RESOURCE_TYPE top
  (* Standard: 61499-2 *)
  (* Version 0.1, 2017-00-25, hpea485, UOA *)
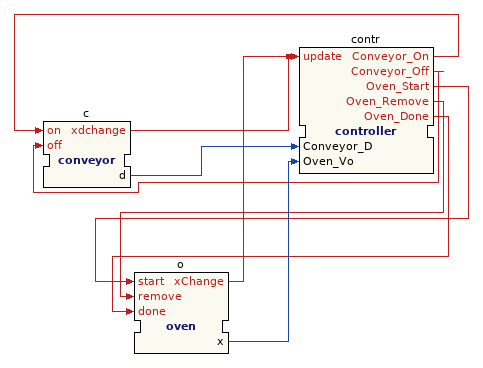
  FBS
    o : oven;
    c : conveyor;
    contr : controller;
  END_FBS
  EVENT_CONNECTIONS
    o.xChange TO contr.update;
    c.xdchange TO contr.update;
    contr.Conveyor_On TO c.on;
    contr.Conveyor_Off TO c.off;
    contr.Oven_Start TO o.start;
    contr.Oven_Remove TO o.remove;
    contr.Oven_Done TO o.done;
  END_CONNECTIONS
  DATA_CONNECTIONS
    o.x TO contr.Oven_Vo;
    c.d TO contr.Conveyor_D;
  END_CONNECTIONS
END_RESOURCE_TYPE
